TYPE ST_DiagnosticCalculations :
STRUCT
	Count		: UDINT;
	Mean		: FLOAT;
	Minimum		: FLOAT;
	Maximum		: FLOAT;
	First		: FLOAT;
	Last		: FLOAT;
	Sum			: FLOAT;
	Variance	: FLOAT;
	Step		: FLOAT;
	Range		: FLOAT;
	StdDev		: FLOAT;
	Difference	: FLOAT;
END_STRUCT
END_TYPE

(* stored: Version 1.1.0.1
   DUT ST_DiagnosticCalculations: Id {7483041e-de20-024f-25aa-723763fa6e7f} *)
